Fanuc KAREL source: kt00380.KL

PROGRAM KT00380
%NOLOCKGROUP
VAR
H1 : ARRAY[2] OF SHORT
R2:REAL
OUT:BOOLEAN
BEGIN
H1[1]=2
R2=3.0
OUT=((H1[1])<=R2)
END KT00380
